PROGRAM MAIN
VAR
END_VAR

END_PROGRAM

(* stored: Version 1.1.0.1
   POU MAIN: Id {d275fa6e-5050-4341-9152-d4fd4111fe0d} *)
